// TwinCAT 3 PLC project SSP_M_EGB_v1
// ProgramVersion: 3.1.4024.0
// libraries:
//   EfficientIO Communicator, * (EfficientIO)
//   EfficientIO Energy Basic, * (EfficientIO)
//   Lynus Persistent Data V1, * (Lynus AG)
//   Lynus Standards, * (EfficientIO)
//   Tc2_Standard, * (Beckhoff Automation GmbH)
//   Tc2_System, * (Beckhoff Automation GmbH)
//   Tc2_Utilities, * (Beckhoff Automation GmbH)
//   Tc3_IPCDiag, * (Beckhoff Automation GmbH)
//   Tc3_Module, * (Beckhoff Automation GmbH)
// project tree:
//   ENUM/ E_State.TcDUT (not stored)
//   / FastTask.TcTTO, MiddleTask.TcTTO, SlowTask.TcTTO
//   FBs/ FB_EM_Beckhoff_KL3403_T.TcPOU, prg_ReadDeviceName.TcPOU (not stored)
//   POUs/ prgCalc.TcPOU, prgComEffIO.TcPOU, prgEM.TcPOU, prgPersistent.TcPOU, prgRWEffIO.TcPOU, prgVarEffIO.TcPOU (not stored)

CONFIGURATION SSP_M_EGB_v1
    RESOURCE PLC ON TwinCAT3
        TASK FastTask(INTERVAL := T#10ms, PRIORITY := 21);
        TASK MiddleTask(INTERVAL := T#10ms, PRIORITY := 23);
        TASK SlowTask(INTERVAL := T#10ms, PRIORITY := 22);
        PROGRAM prgRWEffIO WITH FastTask : prgRWEffIO;
        PROGRAM prgVarEffIO WITH FastTask : prgVarEffIO;
        PROGRAM prgPersistent WITH MiddleTask : prgPersistent;
        PROGRAM prgEM WITH MiddleTask : prgEM;
        PROGRAM prgCalc WITH MiddleTask : prgCalc;
        PROGRAM prgComEffIO WITH SlowTask : prgComEffIO;
    END_RESOURCE
END_CONFIGURATION

// ---- POUs/prgRWEffIO.TcPOU
PROGRAM prgRWEffIO
VAR
	fbRW1		: FB_ReadWrite_V2;
	fbRW2		: FB_ReadWrite;
	fbRW3		: FB_ReadWrite;
END_VAR

fbRW1(	eUploadType := eSelectDataUploadType.e_Change_noIntervall,
		bBusy=> , 
		bError=> , 
		udiErrorCodeOut=> , 
		eErrorReadWrite_Out=> );

fbRW2();
		
fbRW3();

END_PROGRAM

// ---- POUs/prgPersistent.TcPOU
PROGRAM prgPersistent
VAR
	fbUSV		: FB_WritePersistentData_CX81xx;
	
	fb_Reboot		: NT_reboot;
	m_Reboot		: BOOL:=FALSE;
END_VAR

fbUSV(
	eSaveModeData:= eUSVSaveMode.eSaveWhenPowerfail, 
	bLoadPersistentDataOk=> , 
	bPowerFailDetect=> , 
	bError=> , 
	bySaveProcess=> , 
	dwStorageLast24h=> , 
	udiErrorCode=> );
	
	
fb_Reboot(	netid := '',
			delay := 2,
			start := m_Reboot);

END_PROGRAM

// ---- POUs/prgEM.TcPOU
PROGRAM prgEM
VAR	
	fbKBusState		: FB_K_Bus_State;
	
	fbEM1			: FB_EM_Beckhoff_KL3403_T;
	fbEM1Counter	: FB_EnergyCounter;
	
	fbEM2			: FB_EM_Beckhoff_KL3403_T;
	fbEM2Counter	: FB_EnergyCounter;
	
	fbEM3			: FB_EM_Beckhoff_KL3403_T;
	fbEM3Counter	: FB_EnergyCounter;
	
	fbEM4			: FB_EM_Beckhoff_KL3403_T;
	fbEM4Counter	: FB_EnergyCounter;
	
	fbEM5			: FB_EM_Beckhoff_KL3403_T;
	fbEM5Counter	: FB_EnergyCounter;
	
	fbEM6			: FB_EM_Beckhoff_KL3403_T;
	fbEM6Counter	: FB_EnergyCounter;
	
	fbEM7			: FB_EM_Beckhoff_KL3403_T;
	fbEM7Counter	: FB_EnergyCounter;
	
	fbEM8			: FB_EM_Beckhoff_KL3403_T;
	fbEM8Counter	: FB_EnergyCounter;
	
	fbEM9			: FB_EM_Beckhoff_KL3403_T;
	fbEM9Counter	: FB_EnergyCounter;

	//EM1 (CEE32 3phase Measurement)
	lr_RealPower_EM1		: LREAL;					//{#lynus.ag#()}
	lr_ApparentPower_EM1	: LREAL;					//{#lynus.ag#()}
	lr_ReactivePower_EM1	: LREAL;					//{#lynus.ag#()}
	lr_Frequency_EM1		: LREAL;					//{#lynus.ag#()}
    lr_RealPower_EM1_L1		: LREAL;					//{#lynus.ag#()}
    lr_RealPower_EM1_L2		: LREAL;					//{#lynus.ag#()}
    lr_RealPower_EM1_L3		: LREAL;					//{#lynus.ag#()}
	lr_Powerfactor_EM1_L1	: LREAL;					//{#lynus.ag#()}
	lr_Powerfactor_EM1_L2	: LREAL;					//{#lynus.ag#()}
	lr_Powerfactor_EM1_L3	: LREAL;					//{#lynus.ag#()}
	lr_ApparentPower_EM1_L1	: LREAL;					//{#lynus.ag#()}
    lr_ApparentPower_EM1_L2	: LREAL;					//{#lynus.ag#()}
    lr_ApparentPower_EM1_L3	: LREAL;					//{#lynus.ag#()}
	lr_ReactivePower_EM1_L1	: LREAL;					//{#lynus.ag#()}
    lr_ReactivePower_EM1_L2	: LREAL;					//{#lynus.ag#()}
    lr_ReactivePower_EM1_L3	: LREAL;					//{#lynus.ag#()}
	lr_Voltage_EM1_L1N		: LREAL;					//{#lynus.ag#()}
	lr_Voltage_EM1_L2N		: LREAL;					//{#lynus.ag#()}
	lr_Voltage_EM1_L3N		: LREAL;					//{#lynus.ag#()}
	lr_Voltage_EM1_L1L2		: LREAL;					//{#lynus.ag#()}
	lr_Voltage_EM1_L2L3		: LREAL;					//{#lynus.ag#()}
	lr_Voltage_EM1_L3L1		: LREAL;					//{#lynus.ag#()}
 	lr_Current_EM1_L1		: LREAL;					//{#lynus.ag#()}
	lr_Current_EM1_L2		: LREAL;					//{#lynus.ag#()}
	lr_Current_EM1_L3		: LREAL;					//{#lynus.ag#()}

    //EM2 (CEE32 3phase Measurement)
	lr_RealPower_EM2		: LREAL;					//{#lynus.ag#()}
	lr_ApparentPower_EM2	: LREAL;					//{#lynus.ag#()}
	lr_ReactivePower_EM2	: LREAL;					//{#lynus.ag#()}
	lr_Frequency_EM2		: LREAL;					//{#lynus.ag#()}
    lr_RealPower_EM2_L1		: LREAL;					//{#lynus.ag#()}
    lr_RealPower_EM2_L2		: LREAL;					//{#lynus.ag#()}
    lr_RealPower_EM2_L3		: LREAL;					//{#lynus.ag#()}
	lr_Powerfactor_EM2_L1	: LREAL;					//{#lynus.ag#()}
	lr_Powerfactor_EM2_L2	: LREAL;					//{#lynus.ag#()}
	lr_Powerfactor_EM2_L3	: LREAL;					//{#lynus.ag#()}
	lr_ApparentPower_EM2_L1	: LREAL;					//{#lynus.ag#()}
    lr_ApparentPower_EM2_L2	: LREAL;					//{#lynus.ag#()}
    lr_ApparentPower_EM2_L3	: LREAL;					//{#lynus.ag#()}
	lr_ReactivePower_EM2_L1	: LREAL;					//{#lynus.ag#()}
    lr_ReactivePower_EM2_L2	: LREAL;					//{#lynus.ag#()}
    lr_ReactivePower_EM2_L3	: LREAL;					//{#lynus.ag#()}
	lr_Voltage_EM2_L1N		: LREAL;					//{#lynus.ag#()}
	lr_Voltage_EM2_L2N		: LREAL;					//{#lynus.ag#()}
	lr_Voltage_EM2_L3N		: LREAL;					//{#lynus.ag#()}
	lr_Voltage_EM2_L1L2		: LREAL;					//{#lynus.ag#()}
	lr_Voltage_EM2_L2L3		: LREAL;					//{#lynus.ag#()}
	lr_Voltage_EM2_L3L1		: LREAL;					//{#lynus.ag#()}
 	lr_Current_EM2_L1		: LREAL;					//{#lynus.ag#()}
	lr_Current_EM2_L2		: LREAL;					//{#lynus.ag#()}
	lr_Current_EM2_L3		: LREAL;					//{#lynus.ag#()}
	
    //EM3 (CEE32 3phase Measurement)
	lr_RealPower_EM3		: LREAL;					//{#lynus.ag#()}
	lr_ApparentPower_EM3	: LREAL;					//{#lynus.ag#()}
	lr_ReactivePower_EM3	: LREAL;					//{#lynus.ag#()}
	lr_Frequency_EM3		: LREAL;					//{#lynus.ag#()}
    lr_RealPower_EM3_L1		: LREAL;					//{#lynus.ag#()}
    lr_RealPower_EM3_L2		: LREAL;					//{#lynus.ag#()}
    lr_RealPower_EM3_L3		: LREAL;					//{#lynus.ag#()}
	lr_Powerfactor_EM3_L1	: LREAL;					//{#lynus.ag#()}
	lr_Powerfactor_EM3_L2	: LREAL;					//{#lynus.ag#()}
	lr_Powerfactor_EM3_L3	: LREAL;					//{#lynus.ag#()}
	lr_ApparentPower_EM3_L1	: LREAL;					//{#lynus.ag#()}
    lr_ApparentPower_EM3_L2	: LREAL;					//{#lynus.ag#()}
    lr_ApparentPower_EM3_L3	: LREAL;					//{#lynus.ag#()}
	lr_ReactivePower_EM3_L1	: LREAL;					//{#lynus.ag#()}
    lr_ReactivePower_EM3_L2	: LREAL;					//{#lynus.ag#()}
    lr_ReactivePower_EM3_L3	: LREAL;					//{#lynus.ag#()}
	lr_Voltage_EM3_L1N		: LREAL;					//{#lynus.ag#()}
	lr_Voltage_EM3_L2N		: LREAL;					//{#lynus.ag#()}
	lr_Voltage_EM3_L3N		: LREAL;					//{#lynus.ag#()}
	lr_Voltage_EM3_L1L2		: LREAL;					//{#lynus.ag#()}
	lr_Voltage_EM3_L2L3		: LREAL;					//{#lynus.ag#()}
	lr_Voltage_EM3_L3L1		: LREAL;					//{#lynus.ag#()}
 	lr_Current_EM3_L1		: LREAL;					//{#lynus.ag#()}
	lr_Current_EM3_L2		: LREAL;					//{#lynus.ag#()}
	lr_Current_EM3_L3		: LREAL;					//{#lynus.ag#()}

    //EM4 (CEE32 3phase Measurement)
	lr_RealPower_EM4		: LREAL;					//{#lynus.ag#()}
	lr_ApparentPower_EM4	: LREAL;					//{#lynus.ag#()}
	lr_ReactivePower_EM4	: LREAL;					//{#lynus.ag#()}
	lr_Frequency_EM4		: LREAL;					//{#lynus.ag#()}
    lr_RealPower_EM4_L1		: LREAL;					//{#lynus.ag#()}
    lr_RealPower_EM4_L2		: LREAL;					//{#lynus.ag#()}
    lr_RealPower_EM4_L3		: LREAL;					//{#lynus.ag#()}
	lr_Powerfactor_EM4_L1	: LREAL;					//{#lynus.ag#()}
	lr_Powerfactor_EM4_L2	: LREAL;					//{#lynus.ag#()}
	lr_Powerfactor_EM4_L3	: LREAL;					//{#lynus.ag#()}
	lr_ApparentPower_EM4_L1	: LREAL;					//{#lynus.ag#()}
    lr_ApparentPower_EM4_L2	: LREAL;					//{#lynus.ag#()}
    lr_ApparentPower_EM4_L3	: LREAL;					//{#lynus.ag#()}
	lr_ReactivePower_EM4_L1	: LREAL;					//{#lynus.ag#()}
    lr_ReactivePower_EM4_L2	: LREAL;					//{#lynus.ag#()}
    lr_ReactivePower_EM4_L3	: LREAL;					//{#lynus.ag#()}
	lr_Voltage_EM4_L1N		: LREAL;					//{#lynus.ag#()}
	lr_Voltage_EM4_L2N		: LREAL;					//{#lynus.ag#()}
	lr_Voltage_EM4_L3N		: LREAL;					//{#lynus.ag#()}
	lr_Voltage_EM4_L1L2		: LREAL;					//{#lynus.ag#()}
	lr_Voltage_EM4_L2L3		: LREAL;					//{#lynus.ag#()}
	lr_Voltage_EM4_L3L1		: LREAL;					//{#lynus.ag#()}
 	lr_Current_EM4_L1		: LREAL;					//{#lynus.ag#()}
	lr_Current_EM4_L2		: LREAL;					//{#lynus.ag#()}
	lr_Current_EM4_L3		: LREAL;					//{#lynus.ag#()}

    //EM5 (CEE32 3phase Measurement)
	lr_RealPower_EM5		: LREAL;					//{#lynus.ag#()}
	lr_ApparentPower_EM5	: LREAL;					//{#lynus.ag#()}
	lr_ReactivePower_EM5	: LREAL;					//{#lynus.ag#()}
	lr_Frequency_EM5		: LREAL;					//{#lynus.ag#()}
    lr_RealPower_EM5_L1		: LREAL;					//{#lynus.ag#()}
    lr_RealPower_EM5_L2		: LREAL;					//{#lynus.ag#()}
    lr_RealPower_EM5_L3		: LREAL;					//{#lynus.ag#()}
	lr_Powerfactor_EM5_L1	: LREAL;					//{#lynus.ag#()}
	lr_Powerfactor_EM5_L2	: LREAL;					//{#lynus.ag#()}
	lr_Powerfactor_EM5_L3	: LREAL;					//{#lynus.ag#()}
	lr_ApparentPower_EM5_L1	: LREAL;					//{#lynus.ag#()}
    lr_ApparentPower_EM5_L2	: LREAL;					//{#lynus.ag#()}
    lr_ApparentPower_EM5_L3	: LREAL;					//{#lynus.ag#()}
	lr_ReactivePower_EM5_L1	: LREAL;					//{#lynus.ag#()}
    lr_ReactivePower_EM5_L2	: LREAL;					//{#lynus.ag#()}
    lr_ReactivePower_EM5_L3	: LREAL;					//{#lynus.ag#()}
	lr_Voltage_EM5_L1N		: LREAL;					//{#lynus.ag#()}
	lr_Voltage_EM5_L2N		: LREAL;					//{#lynus.ag#()}
	lr_Voltage_EM5_L3N		: LREAL;					//{#lynus.ag#()}
	lr_Voltage_EM5_L1L2		: LREAL;					//{#lynus.ag#()}
	lr_Voltage_EM5_L2L3		: LREAL;					//{#lynus.ag#()}
	lr_Voltage_EM5_L3L1		: LREAL;					//{#lynus.ag#()}
 	lr_Current_EM5_L1		: LREAL;					//{#lynus.ag#()}
	lr_Current_EM5_L2		: LREAL;					//{#lynus.ag#()}
	lr_Current_EM5_L3		: LREAL;					//{#lynus.ag#()}

    //EM6 (CEE32 3phase Measurement)
	lr_RealPower_EM6		: LREAL;					//{#lynus.ag#()}
	lr_ApparentPower_EM6	: LREAL;					//{#lynus.ag#()}
	lr_ReactivePower_EM6	: LREAL;					//{#lynus.ag#()}
	lr_Frequency_EM6		: LREAL;					//{#lynus.ag#()}
    lr_RealPower_EM6_L1		: LREAL;					//{#lynus.ag#()}
    lr_RealPower_EM6_L2		: LREAL;					//{#lynus.ag#()}
    lr_RealPower_EM6_L3		: LREAL;					//{#lynus.ag#()}
	lr_Powerfactor_EM6_L1	: LREAL;					//{#lynus.ag#()}
	lr_Powerfactor_EM6_L2	: LREAL;					//{#lynus.ag#()}
	lr_Powerfactor_EM6_L3	: LREAL;					//{#lynus.ag#()}
	lr_ApparentPower_EM6_L1	: LREAL;					//{#lynus.ag#()}
    lr_ApparentPower_EM6_L2	: LREAL;					//{#lynus.ag#()}
    lr_ApparentPower_EM6_L3	: LREAL;					//{#lynus.ag#()}
	lr_ReactivePower_EM6_L1	: LREAL;					//{#lynus.ag#()}
    lr_ReactivePower_EM6_L2	: LREAL;					//{#lynus.ag#()}
    lr_ReactivePower_EM6_L3	: LREAL;					//{#lynus.ag#()}
	lr_Voltage_EM6_L1N		: LREAL;					//{#lynus.ag#()}
	lr_Voltage_EM6_L2N		: LREAL;					//{#lynus.ag#()}
	lr_Voltage_EM6_L3N		: LREAL;					//{#lynus.ag#()}
	lr_Voltage_EM6_L1L2		: LREAL;					//{#lynus.ag#()}
	lr_Voltage_EM6_L2L3		: LREAL;					//{#lynus.ag#()}
	lr_Voltage_EM6_L3L1		: LREAL;					//{#lynus.ag#()}
 	lr_Current_EM6_L1		: LREAL;					//{#lynus.ag#()}
	lr_Current_EM6_L2		: LREAL;					//{#lynus.ag#()}
	lr_Current_EM6_L3		: LREAL;					//{#lynus.ag#()}

    //EM7 (CEE32 3phase Measurement)
	lr_RealPower_EM7		: LREAL;					//{#lynus.ag#()}
	lr_ApparentPower_EM7	: LREAL;					//{#lynus.ag#()}
	lr_ReactivePower_EM7	: LREAL;					//{#lynus.ag#()}
	lr_Frequency_EM7		: LREAL;					//{#lynus.ag#()}
    lr_RealPower_EM7_L1		: LREAL;					//{#lynus.ag#()}
    lr_RealPower_EM7_L2		: LREAL;					//{#lynus.ag#()}
    lr_RealPower_EM7_L3		: LREAL;					//{#lynus.ag#()}
	lr_Powerfactor_EM7_L1	: LREAL;					//{#lynus.ag#()}
	lr_Powerfactor_EM7_L2	: LREAL;					//{#lynus.ag#()}
	lr_Powerfactor_EM7_L3	: LREAL;					//{#lynus.ag#()}
	lr_ApparentPower_EM7_L1	: LREAL;					//{#lynus.ag#()}
    lr_ApparentPower_EM7_L2	: LREAL;					//{#lynus.ag#()}
    lr_ApparentPower_EM7_L3	: LREAL;					//{#lynus.ag#()}
	lr_ReactivePower_EM7_L1	: LREAL;					//{#lynus.ag#()}
    lr_ReactivePower_EM7_L2	: LREAL;					//{#lynus.ag#()}
    lr_ReactivePower_EM7_L3	: LREAL;					//{#lynus.ag#()}
	lr_Voltage_EM7_L1N		: LREAL;					//{#lynus.ag#()}
	lr_Voltage_EM7_L2N		: LREAL;					//{#lynus.ag#()}
	lr_Voltage_EM7_L3N		: LREAL;					//{#lynus.ag#()}
	lr_Voltage_EM7_L1L2		: LREAL;					//{#lynus.ag#()}
	lr_Voltage_EM7_L2L3		: LREAL;					//{#lynus.ag#()}
	lr_Voltage_EM7_L3L1		: LREAL;					//{#lynus.ag#()}
 	lr_Current_EM7_L1		: LREAL;					//{#lynus.ag#()}
	lr_Current_EM7_L2		: LREAL;					//{#lynus.ag#()}
	lr_Current_EM7_L3		: LREAL;					//{#lynus.ag#()}

    //EM8 (CEE32 3phase Measurement)
	lr_RealPower_EM8		: LREAL;					//{#lynus.ag#()}
	lr_ApparentPower_EM8	: LREAL;					//{#lynus.ag#()}
	lr_ReactivePower_EM8	: LREAL;					//{#lynus.ag#()}
	lr_Frequency_EM8		: LREAL;					//{#lynus.ag#()}
    lr_RealPower_EM8_L1		: LREAL;					//{#lynus.ag#()}
    lr_RealPower_EM8_L2		: LREAL;					//{#lynus.ag#()}
    lr_RealPower_EM8_L3		: LREAL;					//{#lynus.ag#()}
	lr_Powerfactor_EM8_L1	: LREAL;					//{#lynus.ag#()}
	lr_Powerfactor_EM8_L2	: LREAL;					//{#lynus.ag#()}
	lr_Powerfactor_EM8_L3	: LREAL;					//{#lynus.ag#()}
	lr_ApparentPower_EM8_L1	: LREAL;					//{#lynus.ag#()}
    lr_ApparentPower_EM8_L2	: LREAL;					//{#lynus.ag#()}
    lr_ApparentPower_EM8_L3	: LREAL;					//{#lynus.ag#()}
	lr_ReactivePower_EM8_L1	: LREAL;					//{#lynus.ag#()}
    lr_ReactivePower_EM8_L2	: LREAL;					//{#lynus.ag#()}
    lr_ReactivePower_EM8_L3	: LREAL;					//{#lynus.ag#()}
	lr_Voltage_EM8_L1N		: LREAL;					//{#lynus.ag#()}
	lr_Voltage_EM8_L2N		: LREAL;					//{#lynus.ag#()}
	lr_Voltage_EM8_L3N		: LREAL;					//{#lynus.ag#()}
	lr_Voltage_EM8_L1L2		: LREAL;					//{#lynus.ag#()}
	lr_Voltage_EM8_L2L3		: LREAL;					//{#lynus.ag#()}
	lr_Voltage_EM8_L3L1		: LREAL;					//{#lynus.ag#()}
 	lr_Current_EM8_L1		: LREAL;					//{#lynus.ag#()}
	lr_Current_EM8_L2		: LREAL;					//{#lynus.ag#()}
	lr_Current_EM8_L3		: LREAL;					//{#lynus.ag#()}

    //EM9 (CEE32 3phase Measurement)
	lr_RealPower_EM9		: LREAL;					//{#lynus.ag#()}
	lr_ApparentPower_EM9	: LREAL;					//{#lynus.ag#()}
	lr_ReactivePower_EM9	: LREAL;					//{#lynus.ag#()}
	lr_Frequency_EM9		: LREAL;					//{#lynus.ag#()}
    lr_RealPower_EM9_L1		: LREAL;					//{#lynus.ag#()}
    lr_RealPower_EM9_L2		: LREAL;					//{#lynus.ag#()}
    lr_RealPower_EM9_L3		: LREAL;					//{#lynus.ag#()}
	lr_Powerfactor_EM9_L1	: LREAL;					//{#lynus.ag#()}
	lr_Powerfactor_EM9_L2	: LREAL;					//{#lynus.ag#()}
	lr_Powerfactor_EM9_L3	: LREAL;					//{#lynus.ag#()}
	lr_ApparentPower_EM9_L1	: LREAL;					//{#lynus.ag#()}
    lr_ApparentPower_EM9_L2	: LREAL;					//{#lynus.ag#()}
    lr_ApparentPower_EM9_L3	: LREAL;					//{#lynus.ag#()}
	lr_ReactivePower_EM9_L1	: LREAL;					//{#lynus.ag#()}
    lr_ReactivePower_EM9_L2	: LREAL;					//{#lynus.ag#()}
    lr_ReactivePower_EM9_L3	: LREAL;					//{#lynus.ag#()}
	lr_Voltage_EM9_L1N		: LREAL;					//{#lynus.ag#()}
	lr_Voltage_EM9_L2N		: LREAL;					//{#lynus.ag#()}
	lr_Voltage_EM9_L3N		: LREAL;					//{#lynus.ag#()}
	lr_Voltage_EM9_L1L2		: LREAL;					//{#lynus.ag#()}
	lr_Voltage_EM9_L2L3		: LREAL;					//{#lynus.ag#()}
	lr_Voltage_EM9_L3L1		: LREAL;					//{#lynus.ag#()}
 	lr_Current_EM9_L1		: LREAL;					//{#lynus.ag#()}
	lr_Current_EM9_L2		: LREAL;					//{#lynus.ag#()}
	lr_Current_EM9_L3		: LREAL;					//{#lynus.ag#()}
END_VAR

VAR PERSISTENT
	lr_EnergyCounter_EM1	: LREAL;					//{#lynus.ag#()}
	lr_EnergyCounter_EM2	: LREAL;					//{#lynus.ag#()}
    lr_EnergyCounter_EM3	: LREAL;					//{#lynus.ag#()}
    lr_EnergyCounter_EM4	: LREAL;					//{#lynus.ag#()}
    lr_EnergyCounter_EM5	: LREAL;					//{#lynus.ag#()}
    lr_EnergyCounter_EM6	: LREAL;					//{#lynus.ag#()}
    lr_EnergyCounter_EM7	: LREAL;					//{#lynus.ag#()}
    lr_EnergyCounter_EM8	: LREAL;					//{#lynus.ag#()}
    lr_EnergyCounter_EM9	: LREAL;					//{#lynus.ag#()}
END_VAR

fbKBusState(	uiKBusState_OUT=> , 
				b_Kbus_notOk=> , 
				word_ErrorCount=> );

//EM1 (CEE32 3phase Measurement)
fbEM1(
	bEnable:= TRUE, 
	bChannel1Invers:= FALSE,
	bChannel2Invers:= FALSE,
	bChannel3Invers:= FALSE,
	uiCurrentTransformerRatioL1:= 35, 
	uiCurrentTransformerRatioL2:= 35, 
	uiCurrentTransformerRatioL3:= 35, 
	uiKBusState_IN:= fbKBusState.uiKBusState_OUT, 
	stDataEMPower=> , 
	stDataEMCounter=> , 
	stDataEMPowerRealTime=> , 
	stDataEMCounterRealTime=> , 
	diNrOfEM_OUT=> );

lr_RealPower_EM1 := fbEM1.stDataEMPower.lrPowerTotal;
lr_ApparentPower_EM1 := fbEM1.stDataEMPower.lrApparentPowerTotal;
lr_ReactivePower_EM1 := fbEM1.stDataEMPower.lrReactivePowerTotal;
lr_Frequency_EM1 := fbEM1.stDataEMPower.lrFrequency;
lr_RealPower_EM1_L1 := fbEM1.stDataEMPower.lrPowerL1;
lr_RealPower_EM1_L2 := fbEM1.stDataEMPower.lrPowerL2;
lr_RealPower_EM1_L3 := fbEM1.stDataEMPower.lrPowerL3;
lr_Voltage_EM1_L1N := fbEM1.stDataEMPower.lrVoltageL1N;
lr_Voltage_EM1_L2N := fbEM1.stDataEMPower.lrVoltageL2N;
lr_Voltage_EM1_L3N := fbEM1.stDataEMPower.lrVoltageL3N;
lr_Voltage_EM1_L1L2 := fbEM1.stDataEMPower.lrVoltageL1L2;
lr_Voltage_EM1_L2L3 := fbEM1.stDataEMPower.lrVoltageL2L3;
lr_Voltage_EM1_L3L1 := fbEM1.stDataEMPower.lrVoltageL3L1;
lr_Current_EM1_L1 := fbEM1.stDataEMPower.lrCurrentL1;
lr_Current_EM1_L2 := fbEM1.stDataEMPower.lrCurrentL2;
lr_Current_EM1_L3 := fbEM1.stDataEMPower.lrCurrentL3;
lr_Powerfactor_EM1_L1 := fbEM1.lrPowerfactorL1;
lr_Powerfactor_EM1_L2 := fbEM1.lrPowerfactorL2;
lr_Powerfactor_EM1_L3 := fbEM1.lrPowerfactorL3;
(*
lr_ApparentPower_EM1_L1 := fbEM1.lrApparentPowerL1;
lr_ApparentPower_EM1_L2 := fbEM1.lrApparentPowerL2;
lr_ApparentPower_EM1_L3 := fbEM1.lrApparentPowerL3;
lr_ReactivePower_EM1_L1 := fbEM1.lrReactivePowerL1;
lr_ReactivePower_EM1_L2 := fbEM1.lrReactivePowerL2;
lr_ReactivePower_EM1_L3 := fbEM1.lrReactivePowerL3;
*)
fbEM1Counter(
	byActiveTariff:= 1, 
	lrPowerInput:= lr_RealPower_EM1, 
	lrTotalCounterEnergy_Consumption=> , 
	lrTotalCounterEnergy_Production=> , 
	lrCounterEnergyT1_Consumption=> , 
	lrCounterEnergyT2_Consumption=> , 
	lrCounterEnergyT1_Production=> , 
	lrCounterEnergyT2_Production=> );
	
IF fbEM1Counter.lrTotalCounterEnergy_Consumption > lr_EnergyCounter_EM1 THEN  	
	lr_EnergyCounter_EM1 := fbEM1Counter.lrTotalCounterEnergy_Consumption;
END_IF


//EM2 (CEE32 3phase Measurement)
fbEM2(
	bEnable:= TRUE, 
	bChannel1Invers:= FALSE,
	bChannel2Invers:= FALSE,
	bChannel3Invers:= FALSE,
	uiCurrentTransformerRatioL1:= 35, 
	uiCurrentTransformerRatioL2:= 35, 
	uiCurrentTransformerRatioL3:= 35, 
	uiKBusState_IN:= fbKBusState.uiKBusState_OUT, 
	stDataEMPower=> , 
	stDataEMCounter=> , 
	stDataEMPowerRealTime=> , 
	stDataEMCounterRealTime=> , 
	diNrOfEM_OUT=> );

lr_RealPower_EM2 := fbEM2.stDataEMPower.lrPowerTotal;
lr_ApparentPower_EM2 := fbEM2.stDataEMPower.lrApparentPowerTotal;
lr_ReactivePower_EM2 := fbEM2.stDataEMPower.lrReactivePowerTotal;
lr_Frequency_EM2 := fbEM2.stDataEMPower.lrFrequency;
lr_RealPower_EM2_L1 := fbEM2.stDataEMPower.lrPowerL1;
lr_RealPower_EM2_L2 := fbEM2.stDataEMPower.lrPowerL2;
lr_RealPower_EM2_L3 := fbEM2.stDataEMPower.lrPowerL3;
lr_Voltage_EM2_L1N := fbEM2.stDataEMPower.lrVoltageL1N;
lr_Voltage_EM2_L2N := fbEM2.stDataEMPower.lrVoltageL2N;
lr_Voltage_EM2_L3N := fbEM2.stDataEMPower.lrVoltageL3N;
lr_Voltage_EM2_L1L2 := fbEM2.stDataEMPower.lrVoltageL1L2;
lr_Voltage_EM2_L2L3 := fbEM2.stDataEMPower.lrVoltageL2L3;
lr_Voltage_EM2_L3L1 := fbEM2.stDataEMPower.lrVoltageL3L1;
lr_Current_EM2_L1 := fbEM2.stDataEMPower.lrCurrentL1;
lr_Current_EM2_L2 := fbEM2.stDataEMPower.lrCurrentL2;
lr_Current_EM2_L3 := fbEM2.stDataEMPower.lrCurrentL3;
lr_Powerfactor_EM2_L1 := fbEM2.lrPowerfactorL1;
lr_Powerfactor_EM2_L2 := fbEM2.lrPowerfactorL2;
lr_Powerfactor_EM2_L3 := fbEM2.lrPowerfactorL3;
(*
lr_ApparentPower_EM2_L1 := fbEM2.lrApparentPowerL1;
lr_ApparentPower_EM2_L2 := fbEM2.lrApparentPowerL2;
lr_ApparentPower_EM2_L3 := fbEM2.lrApparentPowerL3;
lr_ReactivePower_EM2_L1 := fbEM2.lrReactivePowerL1;
lr_ReactivePower_EM2_L2 := fbEM2.lrReactivePowerL2;
lr_ReactivePower_EM2_L3 := fbEM2.lrReactivePowerL3;
*)
fbEM2Counter(
	byActiveTariff:= 1, 
	lrPowerInput:= lr_RealPower_EM2, 
	lrTotalCounterEnergy_Consumption=> , 
	lrTotalCounterEnergy_Production=> , 
	lrCounterEnergyT1_Consumption=> , 
	lrCounterEnergyT2_Consumption=> , 
	lrCounterEnergyT1_Production=> , 
	lrCounterEnergyT2_Production=> );
	
IF fbEM2Counter.lrTotalCounterEnergy_Consumption > lr_EnergyCounter_EM2 THEN  	
	lr_EnergyCounter_EM2 := fbEM2Counter.lrTotalCounterEnergy_Consumption;
END_IF

//EM3 (CEE32 3phase Measurement)
fbEM3(
	bEnable:= TRUE, 
	bChannel1Invers:= FALSE,
	bChannel2Invers:= FALSE,
	bChannel3Invers:= FALSE,
	uiCurrentTransformerRatioL1:= 35, 
	uiCurrentTransformerRatioL2:= 35, 
	uiCurrentTransformerRatioL3:= 35, 
	uiKBusState_IN:= fbKBusState.uiKBusState_OUT, 
	stDataEMPower=> , 
	stDataEMCounter=> , 
	stDataEMPowerRealTime=> , 
	stDataEMCounterRealTime=> , 
	diNrOfEM_OUT=> );

lr_RealPower_EM3 := fbEM3.stDataEMPower.lrPowerTotal;
lr_ApparentPower_EM3 := fbEM3.stDataEMPower.lrApparentPowerTotal;
lr_ReactivePower_EM3 := fbEM3.stDataEMPower.lrReactivePowerTotal;
lr_Frequency_EM3 := fbEM3.stDataEMPower.lrFrequency;
lr_RealPower_EM3_L1 := fbEM3.stDataEMPower.lrPowerL1;
lr_RealPower_EM3_L2 := fbEM3.stDataEMPower.lrPowerL2;
lr_RealPower_EM3_L3 := fbEM3.stDataEMPower.lrPowerL3;
lr_Voltage_EM3_L1N := fbEM3.stDataEMPower.lrVoltageL1N;
lr_Voltage_EM3_L2N := fbEM3.stDataEMPower.lrVoltageL2N;
lr_Voltage_EM3_L3N := fbEM3.stDataEMPower.lrVoltageL3N;
lr_Voltage_EM3_L1L2 := fbEM3.stDataEMPower.lrVoltageL1L2;
lr_Voltage_EM3_L2L3 := fbEM3.stDataEMPower.lrVoltageL2L3;
lr_Voltage_EM3_L3L1 := fbEM3.stDataEMPower.lrVoltageL3L1;
lr_Current_EM3_L1 := fbEM3.stDataEMPower.lrCurrentL1;
lr_Current_EM3_L2 := fbEM3.stDataEMPower.lrCurrentL2;
lr_Current_EM3_L3 := fbEM3.stDataEMPower.lrCurrentL3;
lr_Powerfactor_EM3_L1 := fbEM3.lrPowerfactorL1;
lr_Powerfactor_EM3_L2 := fbEM3.lrPowerfactorL2;
lr_Powerfactor_EM3_L3 := fbEM3.lrPowerfactorL3;
(*
lr_ApparentPower_EM3_L1 := fbEM3.lrApparentPowerL1;
lr_ApparentPower_EM3_L2 := fbEM3.lrApparentPowerL2;
lr_ApparentPower_EM3_L3 := fbEM3.lrApparentPowerL3;
lr_ReactivePower_EM3_L1 := fbEM3.lrReactivePowerL1;
lr_ReactivePower_EM3_L2 := fbEM3.lrReactivePowerL2;
lr_ReactivePower_EM3_L3 := fbEM3.lrReactivePowerL3;
*)
fbEM3Counter(
	byActiveTariff:= 1, 
	lrPowerInput:= lr_RealPower_EM3, 
	lrTotalCounterEnergy_Consumption=> , 
	lrTotalCounterEnergy_Production=> , 
	lrCounterEnergyT1_Consumption=> , 
	lrCounterEnergyT2_Consumption=> , 
	lrCounterEnergyT1_Production=> , 
	lrCounterEnergyT2_Production=> );
	
IF fbEM3Counter.lrTotalCounterEnergy_Consumption > lr_EnergyCounter_EM3 THEN  	
	lr_EnergyCounter_EM3 := fbEM3Counter.lrTotalCounterEnergy_Consumption;
END_IF

//EM4 (CEE32 3phase Measurement)
fbEM4(
	bEnable:= TRUE, 
	bChannel1Invers:= FALSE,
	bChannel2Invers:= FALSE,
	bChannel3Invers:= FALSE,
	uiCurrentTransformerRatioL1:= 35, 
	uiCurrentTransformerRatioL2:= 35, 
	uiCurrentTransformerRatioL3:= 35, 
	uiKBusState_IN:= fbKBusState.uiKBusState_OUT, 
	stDataEMPower=> , 
	stDataEMCounter=> , 
	stDataEMPowerRealTime=> , 
	stDataEMCounterRealTime=> , 
	diNrOfEM_OUT=> );

lr_RealPower_EM4 := fbEM4.stDataEMPower.lrPowerTotal;
lr_ApparentPower_EM4 := fbEM4.stDataEMPower.lrApparentPowerTotal;
lr_ReactivePower_EM4 := fbEM4.stDataEMPower.lrReactivePowerTotal;
lr_Frequency_EM4 := fbEM4.stDataEMPower.lrFrequency;
lr_RealPower_EM4_L1 := fbEM4.stDataEMPower.lrPowerL1;
lr_RealPower_EM4_L2 := fbEM4.stDataEMPower.lrPowerL2;
lr_RealPower_EM4_L3 := fbEM4.stDataEMPower.lrPowerL3;
lr_Voltage_EM4_L1N := fbEM4.stDataEMPower.lrVoltageL1N;
lr_Voltage_EM4_L2N := fbEM4.stDataEMPower.lrVoltageL2N;
lr_Voltage_EM4_L3N := fbEM4.stDataEMPower.lrVoltageL3N;
lr_Voltage_EM4_L1L2 := fbEM4.stDataEMPower.lrVoltageL1L2;
lr_Voltage_EM4_L2L3 := fbEM4.stDataEMPower.lrVoltageL2L3;
lr_Voltage_EM4_L3L1 := fbEM4.stDataEMPower.lrVoltageL3L1;
lr_Current_EM4_L1 := fbEM4.stDataEMPower.lrCurrentL1;
lr_Current_EM4_L2 := fbEM4.stDataEMPower.lrCurrentL2;
lr_Current_EM4_L3 := fbEM4.stDataEMPower.lrCurrentL3;
lr_Powerfactor_EM4_L1 := fbEM4.lrPowerfactorL1;
lr_Powerfactor_EM4_L2 := fbEM4.lrPowerfactorL2;
lr_Powerfactor_EM4_L3 := fbEM4.lrPowerfactorL3;
(*
lr_ApparentPower_EM4_L1 := fbEM4.lrApparentPowerL1;
lr_ApparentPower_EM4_L2 := fbEM4.lrApparentPowerL2;
lr_ApparentPower_EM4_L3 := fbEM4.lrApparentPowerL3;
lr_ReactivePower_EM4_L1 := fbEM4.lrReactivePowerL1;
lr_ReactivePower_EM4_L2 := fbEM4.lrReactivePowerL2;
lr_ReactivePower_EM4_L3 := fbEM4.lrReactivePowerL3;
*)
fbEM4Counter(
	byActiveTariff:= 1, 
	lrPowerInput:= lr_RealPower_EM4, 
	lrTotalCounterEnergy_Consumption=> , 
	lrTotalCounterEnergy_Production=> , 
	lrCounterEnergyT1_Consumption=> , 
	lrCounterEnergyT2_Consumption=> , 
	lrCounterEnergyT1_Production=> , 
	lrCounterEnergyT2_Production=> );
	
IF fbEM4Counter.lrTotalCounterEnergy_Consumption > lr_EnergyCounter_EM4 THEN  	
	lr_EnergyCounter_EM4 := fbEM4Counter.lrTotalCounterEnergy_Consumption;
END_IF

//EM5 (CEE32 3phase Measurement)
fbEM5(
	bEnable:= TRUE, 
	bChannel1Invers:= FALSE,
	bChannel2Invers:= FALSE,
	bChannel3Invers:= FALSE,
	uiCurrentTransformerRatioL1:= 35, 
	uiCurrentTransformerRatioL2:= 35, 
	uiCurrentTransformerRatioL3:= 35, 
	uiKBusState_IN:= fbKBusState.uiKBusState_OUT, 
	stDataEMPower=> , 
	stDataEMCounter=> , 
	stDataEMPowerRealTime=> , 
	stDataEMCounterRealTime=> , 
	diNrOfEM_OUT=> );

lr_RealPower_EM5 := fbEM5.stDataEMPower.lrPowerTotal;
lr_ApparentPower_EM5 := fbEM5.stDataEMPower.lrApparentPowerTotal;
lr_ReactivePower_EM5 := fbEM5.stDataEMPower.lrReactivePowerTotal;
lr_Frequency_EM5 := fbEM5.stDataEMPower.lrFrequency;
lr_RealPower_EM5_L1 := fbEM5.stDataEMPower.lrPowerL1;
lr_RealPower_EM5_L2 := fbEM5.stDataEMPower.lrPowerL2;
lr_RealPower_EM5_L3 := fbEM5.stDataEMPower.lrPowerL3;
lr_Voltage_EM5_L1N := fbEM5.stDataEMPower.lrVoltageL1N;
lr_Voltage_EM5_L2N := fbEM5.stDataEMPower.lrVoltageL2N;
lr_Voltage_EM5_L3N := fbEM5.stDataEMPower.lrVoltageL3N;
lr_Voltage_EM5_L1L2 := fbEM5.stDataEMPower.lrVoltageL1L2;
lr_Voltage_EM5_L2L3 := fbEM5.stDataEMPower.lrVoltageL2L3;
lr_Voltage_EM5_L3L1 := fbEM5.stDataEMPower.lrVoltageL3L1;
lr_Current_EM5_L1 := fbEM5.stDataEMPower.lrCurrentL1;
lr_Current_EM5_L2 := fbEM5.stDataEMPower.lrCurrentL2;
lr_Current_EM5_L3 := fbEM5.stDataEMPower.lrCurrentL3;
lr_Powerfactor_EM5_L1 := fbEM5.lrPowerfactorL1;
lr_Powerfactor_EM5_L2 := fbEM5.lrPowerfactorL2;
lr_Powerfactor_EM5_L3 := fbEM5.lrPowerfactorL3;
(*
lr_ApparentPower_EM5_L1 := fbEM5.lrApparentPowerL1;
lr_ApparentPower_EM5_L2 := fbEM5.lrApparentPowerL2;
lr_ApparentPower_EM5_L3 := fbEM5.lrApparentPowerL3;
lr_ReactivePower_EM5_L1 := fbEM5.lrReactivePowerL1;
lr_ReactivePower_EM5_L2 := fbEM5.lrReactivePowerL2;
lr_ReactivePower_EM5_L3 := fbEM5.lrReactivePowerL3;
*)
fbEM5Counter(
	byActiveTariff:= 1, 
	lrPowerInput:= lr_RealPower_EM5, 
	lrTotalCounterEnergy_Consumption=> , 
	lrTotalCounterEnergy_Production=> , 
	lrCounterEnergyT1_Consumption=> , 
	lrCounterEnergyT2_Consumption=> , 
	lrCounterEnergyT1_Production=> , 
	lrCounterEnergyT2_Production=> );
	
IF fbEM5Counter.lrTotalCounterEnergy_Consumption > lr_EnergyCounter_EM5 THEN  	
	lr_EnergyCounter_EM5 := fbEM5Counter.lrTotalCounterEnergy_Consumption;
END_IF

//EM6 (CEE32 3phase Measurement)
fbEM6(
	bEnable:= TRUE, 
	bChannel1Invers:= FALSE,
	bChannel2Invers:= FALSE,
	bChannel3Invers:= FALSE,
	uiCurrentTransformerRatioL1:= 35, 
	uiCurrentTransformerRatioL2:= 35, 
	uiCurrentTransformerRatioL3:= 35, 
	uiKBusState_IN:= fbKBusState.uiKBusState_OUT, 
	stDataEMPower=> , 
	stDataEMCounter=> , 
	stDataEMPowerRealTime=> , 
	stDataEMCounterRealTime=> , 
	diNrOfEM_OUT=> );

lr_RealPower_EM6 := fbEM6.stDataEMPower.lrPowerTotal;
lr_ApparentPower_EM6 := fbEM6.stDataEMPower.lrApparentPowerTotal;
lr_ReactivePower_EM6 := fbEM6.stDataEMPower.lrReactivePowerTotal;
lr_Frequency_EM6 := fbEM6.stDataEMPower.lrFrequency;
lr_RealPower_EM6_L1 := fbEM6.stDataEMPower.lrPowerL1;
lr_RealPower_EM6_L2 := fbEM6.stDataEMPower.lrPowerL2;
lr_RealPower_EM6_L3 := fbEM6.stDataEMPower.lrPowerL3;
lr_Voltage_EM6_L1N := fbEM6.stDataEMPower.lrVoltageL1N;
lr_Voltage_EM6_L2N := fbEM6.stDataEMPower.lrVoltageL2N;
lr_Voltage_EM6_L3N := fbEM6.stDataEMPower.lrVoltageL3N;
lr_Voltage_EM6_L1L2 := fbEM6.stDataEMPower.lrVoltageL1L2;
lr_Voltage_EM6_L2L3 := fbEM6.stDataEMPower.lrVoltageL2L3;
lr_Voltage_EM6_L3L1 := fbEM6.stDataEMPower.lrVoltageL3L1;
lr_Current_EM6_L1 := fbEM6.stDataEMPower.lrCurrentL1;
lr_Current_EM6_L2 := fbEM6.stDataEMPower.lrCurrentL2;
lr_Current_EM6_L3 := fbEM6.stDataEMPower.lrCurrentL3;
lr_Powerfactor_EM6_L1 := fbEM6.lrPowerfactorL1;
lr_Powerfactor_EM6_L2 := fbEM6.lrPowerfactorL2;
lr_Powerfactor_EM6_L3 := fbEM6.lrPowerfactorL3;
(*
lr_ApparentPower_EM6_L1 := fbEM6.lrApparentPowerL1;
lr_ApparentPower_EM6_L2 := fbEM6.lrApparentPowerL2;
lr_ApparentPower_EM6_L3 := fbEM6.lrApparentPowerL3;
lr_ReactivePower_EM6_L1 := fbEM6.lrReactivePowerL1;
lr_ReactivePower_EM6_L2 := fbEM6.lrReactivePowerL2;
lr_ReactivePower_EM6_L3 := fbEM6.lrReactivePowerL3;
*)
fbEM6Counter(
	byActiveTariff:= 1, 
	lrPowerInput:= lr_RealPower_EM6, 
	lrTotalCounterEnergy_Consumption=> , 
	lrTotalCounterEnergy_Production=> , 
	lrCounterEnergyT1_Consumption=> , 
	lrCounterEnergyT2_Consumption=> , 
	lrCounterEnergyT1_Production=> , 
	lrCounterEnergyT2_Production=> );
	
IF fbEM6Counter.lrTotalCounterEnergy_Consumption > lr_EnergyCounter_EM6 THEN  	
	lr_EnergyCounter_EM6 := fbEM6Counter.lrTotalCounterEnergy_Consumption;
END_IF

//EM7 (CEE32 3phase Measurement)
fbEM7(
	bEnable:= TRUE, 
	bChannel1Invers:= FALSE,
	bChannel2Invers:= FALSE,
	bChannel3Invers:= FALSE,
	uiCurrentTransformerRatioL1:= 35, 
	uiCurrentTransformerRatioL2:= 35, 
	uiCurrentTransformerRatioL3:= 35, 
	uiKBusState_IN:= fbKBusState.uiKBusState_OUT, 
	stDataEMPower=> , 
	stDataEMCounter=> , 
	stDataEMPowerRealTime=> , 
	stDataEMCounterRealTime=> , 
	diNrOfEM_OUT=> );

lr_RealPower_EM7 := fbEM7.stDataEMPower.lrPowerTotal;
lr_ApparentPower_EM7 := fbEM7.stDataEMPower.lrApparentPowerTotal;
lr_ReactivePower_EM7 := fbEM7.stDataEMPower.lrReactivePowerTotal;
lr_Frequency_EM7 := fbEM7.stDataEMPower.lrFrequency;
lr_RealPower_EM7_L1 := fbEM7.stDataEMPower.lrPowerL1;
lr_RealPower_EM7_L2 := fbEM7.stDataEMPower.lrPowerL2;
lr_RealPower_EM7_L3 := fbEM7.stDataEMPower.lrPowerL3;
lr_Voltage_EM7_L1N := fbEM7.stDataEMPower.lrVoltageL1N;
lr_Voltage_EM7_L2N := fbEM7.stDataEMPower.lrVoltageL2N;
lr_Voltage_EM7_L3N := fbEM7.stDataEMPower.lrVoltageL3N;
lr_Voltage_EM7_L1L2 := fbEM7.stDataEMPower.lrVoltageL1L2;
lr_Voltage_EM7_L2L3 := fbEM7.stDataEMPower.lrVoltageL2L3;
lr_Voltage_EM7_L3L1 := fbEM7.stDataEMPower.lrVoltageL3L1;
lr_Current_EM7_L1 := fbEM7.stDataEMPower.lrCurrentL1;
lr_Current_EM7_L2 := fbEM7.stDataEMPower.lrCurrentL2;
lr_Current_EM7_L3 := fbEM7.stDataEMPower.lrCurrentL3;
lr_Powerfactor_EM7_L1 := fbEM7.lrPowerfactorL1;
lr_Powerfactor_EM7_L2 := fbEM7.lrPowerfactorL2;
lr_Powerfactor_EM7_L3 := fbEM7.lrPowerfactorL3;
(*
lr_ApparentPower_EM7_L1 := fbEM7.lrApparentPowerL1;
lr_ApparentPower_EM7_L2 := fbEM7.lrApparentPowerL2;
lr_ApparentPower_EM7_L3 := fbEM7.lrApparentPowerL3;
lr_ReactivePower_EM7_L1 := fbEM7.lrReactivePowerL1;
lr_ReactivePower_EM7_L2 := fbEM7.lrReactivePowerL2;
lr_ReactivePower_EM7_L3 := fbEM7.lrReactivePowerL3;
*)
fbEM7Counter(
	byActiveTariff:= 1, 
	lrPowerInput:= lr_RealPower_EM7, 
	lrTotalCounterEnergy_Consumption=> , 
	lrTotalCounterEnergy_Production=> , 
	lrCounterEnergyT1_Consumption=> , 
	lrCounterEnergyT2_Consumption=> , 
	lrCounterEnergyT1_Production=> , 
	lrCounterEnergyT2_Production=> );
	
IF fbEM7Counter.lrTotalCounterEnergy_Consumption > lr_EnergyCounter_EM7 THEN  	
	lr_EnergyCounter_EM7 := fbEM7Counter.lrTotalCounterEnergy_Consumption;
END_IF

//EM8 (CEE32 3phase Measurement)
fbEM8(
	bEnable:= TRUE, 
	bChannel1Invers:= FALSE,
	bChannel2Invers:= FALSE,
	bChannel3Invers:= FALSE,
	uiCurrentTransformerRatioL1:= 35, 
	uiCurrentTransformerRatioL2:= 35, 
	uiCurrentTransformerRatioL3:= 35, 
	uiKBusState_IN:= fbKBusState.uiKBusState_OUT, 
	stDataEMPower=> , 
	stDataEMCounter=> , 
	stDataEMPowerRealTime=> , 
	stDataEMCounterRealTime=> , 
	diNrOfEM_OUT=> );

lr_RealPower_EM8 := fbEM8.stDataEMPower.lrPowerTotal;
lr_ApparentPower_EM8 := fbEM8.stDataEMPower.lrApparentPowerTotal;
lr_ReactivePower_EM8 := fbEM8.stDataEMPower.lrReactivePowerTotal;
lr_Frequency_EM8 := fbEM8.stDataEMPower.lrFrequency;
lr_RealPower_EM8_L1 := fbEM8.stDataEMPower.lrPowerL1;
lr_RealPower_EM8_L2 := fbEM8.stDataEMPower.lrPowerL2;
lr_RealPower_EM8_L3 := fbEM8.stDataEMPower.lrPowerL3;
lr_Voltage_EM8_L1N := fbEM8.stDataEMPower.lrVoltageL1N;
lr_Voltage_EM8_L2N := fbEM8.stDataEMPower.lrVoltageL2N;
lr_Voltage_EM8_L3N := fbEM8.stDataEMPower.lrVoltageL3N;
lr_Voltage_EM8_L1L2 := fbEM8.stDataEMPower.lrVoltageL1L2;
lr_Voltage_EM8_L2L3 := fbEM8.stDataEMPower.lrVoltageL2L3;
lr_Voltage_EM8_L3L1 := fbEM8.stDataEMPower.lrVoltageL3L1;
lr_Current_EM8_L1 := fbEM8.stDataEMPower.lrCurrentL1;
lr_Current_EM8_L2 := fbEM8.stDataEMPower.lrCurrentL2;
lr_Current_EM8_L3 := fbEM8.stDataEMPower.lrCurrentL3;
lr_Powerfactor_EM8_L1 := fbEM8.lrPowerfactorL1;
lr_Powerfactor_EM8_L2 := fbEM8.lrPowerfactorL2;
lr_Powerfactor_EM8_L3 := fbEM8.lrPowerfactorL3;
(*
lr_ApparentPower_EM8_L1 := fbEM8.lrApparentPowerL1;
lr_ApparentPower_EM8_L2 := fbEM8.lrApparentPowerL2;
lr_ApparentPower_EM8_L3 := fbEM8.lrApparentPowerL3;
lr_ReactivePower_EM8_L1 := fbEM8.lrReactivePowerL1;
lr_ReactivePower_EM8_L2 := fbEM8.lrReactivePowerL2;
lr_ReactivePower_EM8_L3 := fbEM8.lrReactivePowerL3;
*)
fbEM8Counter(
	byActiveTariff:= 1, 
	lrPowerInput:= lr_RealPower_EM8, 
	lrTotalCounterEnergy_Consumption=> , 
	lrTotalCounterEnergy_Production=> , 
	lrCounterEnergyT1_Consumption=> , 
	lrCounterEnergyT2_Consumption=> , 
	lrCounterEnergyT1_Production=> , 
	lrCounterEnergyT2_Production=> );
	
IF fbEM8Counter.lrTotalCounterEnergy_Consumption > lr_EnergyCounter_EM8 THEN  	
	lr_EnergyCounter_EM8 := fbEM8Counter.lrTotalCounterEnergy_Consumption;
END_IF

//EM9 (CEE32 3phase Measurement)
fbEM9(
	bEnable:= TRUE, 
	bChannel1Invers:= FALSE,
	bChannel2Invers:= FALSE,
	bChannel3Invers:= FALSE,
	uiCurrentTransformerRatioL1:= 35, 
	uiCurrentTransformerRatioL2:= 35, 
	uiCurrentTransformerRatioL3:= 35, 
	uiKBusState_IN:= fbKBusState.uiKBusState_OUT, 
	stDataEMPower=> , 
	stDataEMCounter=> , 
	stDataEMPowerRealTime=> , 
	stDataEMCounterRealTime=> , 
	diNrOfEM_OUT=> );

lr_RealPower_EM9 := fbEM9.stDataEMPower.lrPowerTotal;
lr_ApparentPower_EM9 := fbEM9.stDataEMPower.lrApparentPowerTotal;
lr_ReactivePower_EM9 := fbEM9.stDataEMPower.lrReactivePowerTotal;
lr_Frequency_EM9 := fbEM9.stDataEMPower.lrFrequency;
lr_RealPower_EM9_L1 := fbEM9.stDataEMPower.lrPowerL1;
lr_RealPower_EM9_L2 := fbEM9.stDataEMPower.lrPowerL2;
lr_RealPower_EM9_L3 := fbEM9.stDataEMPower.lrPowerL3;
lr_Voltage_EM9_L1N := fbEM9.stDataEMPower.lrVoltageL1N;
lr_Voltage_EM9_L2N := fbEM9.stDataEMPower.lrVoltageL2N;
lr_Voltage_EM9_L3N := fbEM9.stDataEMPower.lrVoltageL3N;
lr_Voltage_EM9_L1L2 := fbEM9.stDataEMPower.lrVoltageL1L2;
lr_Voltage_EM9_L2L3 := fbEM9.stDataEMPower.lrVoltageL2L3;
lr_Voltage_EM9_L3L1 := fbEM9.stDataEMPower.lrVoltageL3L1;
lr_Current_EM9_L1 := fbEM9.stDataEMPower.lrCurrentL1;
lr_Current_EM9_L2 := fbEM9.stDataEMPower.lrCurrentL2;
lr_Current_EM9_L3 := fbEM9.stDataEMPower.lrCurrentL3;
lr_Powerfactor_EM9_L1 := fbEM9.lrPowerfactorL1;
lr_Powerfactor_EM9_L2 := fbEM9.lrPowerfactorL2;
lr_Powerfactor_EM9_L3 := fbEM9.lrPowerfactorL3;
(*
lr_ApparentPower_EM9_L1 := fbEM9.lrApparentPowerL1;
lr_ApparentPower_EM9_L2 := fbEM9.lrApparentPowerL2;
lr_ApparentPower_EM9_L3 := fbEM9.lrApparentPowerL3;
lr_ReactivePower_EM9_L1 := fbEM9.lrReactivePowerL1;
lr_ReactivePower_EM9_L2 := fbEM9.lrReactivePowerL2;
lr_ReactivePower_EM9_L3 := fbEM9.lrReactivePowerL3;
*)
fbEM9Counter(
	byActiveTariff:= 1, 
	lrPowerInput:= lr_RealPower_EM9, 
	lrTotalCounterEnergy_Consumption=> , 
	lrTotalCounterEnergy_Production=> , 
	lrCounterEnergyT1_Consumption=> , 
	lrCounterEnergyT2_Consumption=> , 
	lrCounterEnergyT1_Production=> , 
	lrCounterEnergyT2_Production=> );
	
IF fbEM9Counter.lrTotalCounterEnergy_Consumption > lr_EnergyCounter_EM9 THEN  	
	lr_EnergyCounter_EM9 := fbEM9Counter.lrTotalCounterEnergy_Consumption;
END_IF

END_PROGRAM

// ---- FBs/FB_EM_Beckhoff_KL3403_T.TcPOU
FUNCTION_BLOCK FB_EM_Beckhoff_KL3403_T
VAR_INPUT PERSISTENT
	bEnable							: BOOL;											//Enable the function
	bChannel1Invers					: BOOL;											//Invert the Output data from Channel 1. = L1
	bChannel2Invers					: BOOL;											//Invert the Output data from Channel 2. = L2
	bChannel3Invers					: BOOL;											//Invert the Output data from Channel 3. = L3
	uiCurrentTransformerRatioL1		: UINT;											//Current Transformer Ratio for Channel 1 (L1)
	uiCurrentTransformerRatioL2		: UINT;											//Current Transformer Ratio for Channel 2 (L2)
	uiCurrentTransformerRatioL3		: UINT;											//Current Transformer Ratio for Channel 3 (L3)
END_VAR
VAR_INPUT
	uiKBusState_IN					: UINT;											//K-Bus State from the K-Bus Box on wich the Terminal is connected. (Connect with FB_K_Bus_state)
END_VAR
VAR_OUTPUT
	stDataEMPower					: ST_ElectricMeter_Output_Power;				//Output structure with Data from Electric Meter (Power Data)
	stDataEMCounter					: ST_ElectricMeter_Output_Counter;				//Output structure with Data from Electric Meter (Counter Data)
	stDataEMPowerRealTime			: ST_ElectricMeter_Output_Power;				//Output structure with Data from Electric Meter (Power Data RealTime)
	stDataEMCounterRealTime			: ST_ElectricMeter_Output_Counter;				//Output structure with Data from Electric Meter (Counter Data RealTime)
	diNrOfEM_OUT					: DINT;											//Active Number from the Electric Meter for using on other functions
	lrPowerfactorL1					: LREAL;
	lrPowerfactorL2					: LREAL;
	lrPowerfactorL3					: LREAL;
	lrApparentPowerL1				: LREAL;
	lrApparentPowerL2				: LREAL;
	lrApparentPowerL3				: LREAL;
	lrReactivePowerL1				: LREAL;
	lrReactivePowerL2				: LREAL;
	lrReactivePowerL3				: LREAL;
END_VAR
VAR
	{attribute 'conditionalshow'}
	fbEM							: FB_ElectricMeter;								//Electric Meter Function
	{attribute 'conditionalshow'}
	fbEnergyCounter					: FB_EnergyCounter;								//FB energy Counter, because the KL3403 has no nice logic for the Energy value
	{attribute 'hide'}
	fbNumberDevice					: FB_NumberOfDevice;							//Function block to calcualte the number of the Device
	fbKL3403						: FB_KL3403_SimpleProcessImage;					//Function KL3403
	{attribute 'hide'}
	stDataL1						: ST_KL3403;									//Data from Channel 1 (L1)
	{attribute 'hide'}
	stDataL2						: ST_KL3403;									//Data from Channel 2 (L2)
	{attribute 'hide'}
	stDataL3						: ST_KL3403;									//Data from Channel 3 (L3)
	{attribute 'hide'}
	timDissableFunctions			: TON;											//Timer to dissable the Function after Lynus_Standards.Constants_General.tTimeDissableLynusFunctions Days without connection to the Lynus Cloud
	{attribute 'hide'}
	timResetConnectionOnGVL			: TON;											//Timer to try reset the connection Flag on the GVL. (When somebody delete the Connection Function and make only a onlinechange)
	{attribute 'hide'}
	timSetCounterValues				: TON;											//Timer to set the counter values from the KL3403 Function to the EM Function
	{attribute 'hide'}
	arrPD							: ARRAY[1..7] OF FB_PersistentData_Number;		//Function to save persistent data
	{attribute 'hide'}
	byWaitInStep					: BYTE;											//Wait in Step before start to clean data on PLC
	{attribute 'hide'}
	iStateGVLData					: INT;											//State machine to handle the data on the GVL
	{attribute 'hide'}
	diCounterForGVL					: DINT;											//Counter to clean old data on GVL
END_VAR

//Creator : Kai Ebensperger
//Company : Lynus AG
//Date : 04.10.2021
//Version : 1.0.0.0

//Stefan: Addes S and Q calculation

//With this function is possible to read out all Information from a KL3403
//This Function support only the Simple Process Image and the Ratio in the Terminal register must be Set allways to 1.

//NOTE for diNr.....Designation => 
//_IN = Here Data come in from other Functions or go out to other functions about the GVL
//_OUT = Here Data go out to other functions about the GVL

(*-------------------------------------------------------------Calcualte the number of EM---------------------------------------------------------------*)

fbNumberDevice(
	diActualNumberOfDevices:= Lynus_Standards.GVL_Energy.stNumberOfDevices.diNumberOfElectricMeters, 
	diMaxNumberOfDevices:= Constants_Energy.diMaxNumberOfElectricMeters, 
	udiCounterOnlineChange:= TwinCAT_SystemInfoVarList._AppInfo.OnlineChangeCnt, 
	bNumberIsCalculatet=> , 
	bFPNumberIsCalculatet=> , 
	bOnlineChange=> , 
	diNumberForThisDevice=> diNrOfEM_OUT, 
	diNumberOfTotalDevices=> );

//Write new Numer on GVL
IF fbNumberDevice.bFPNumberIsCalculatet THEN
	Lynus_Standards.GVL_Energy.stNumberOfDevices.diNumberOfElectricMeters := fbNumberDevice.diNumberOfTotalDevices;	
END_IF

//Delete old Number on GVL
IF fbNumberDevice.bOnlineChange THEN 
	Lynus_Standards.GVL_Energy.stNumberOfDevices.diNumberOfElectricMeters := diNrOfEM_OUT;	
		iStateGVLData := 1; 
END_IF

(*-------------------------------------------------------------Service from Backend is ready and check the connection to backen for dissabel/enable Function---------------------------------------------------------------*)

//Try to reset the variable for connection on the GVL. When all is normal then the Lynus Mqtt connection function set this variable to true in the next cycle
//When we have no connection to the backend then after Lynus_Standards.Constants_General.tTimeDissableLynusFunctions days the Function is dissabled with all of his functionalities
timResetConnectionOnGVL(IN:= NOT timResetConnectionOnGVL.Q, PT:= T#1H, Q=> , ET=> );
	IF timResetConnectionOnGVL.Q THEN Lynus_Standards.GVL_Communicator.bStateConnectionToEnableFunctions := FALSE; END_IF
		IF NOT Lynus_Standards.GVL_Communicator.bStateConnectionToEnableFunctions THEN timDissableFunctions.IN := TRUE; ELSE timDissableFunctions.IN := FALSE; END_IF  
			timDissableFunctions(IN:= , PT:= Lynus_Standards.Constants_General.tTimeDissableLynusFunctions, Q=> , ET=> );

(*----------------------------------------------------------------------------------------KL3403 Communication----------------------------------------------------------------------------------------------*)

fbKL3403(
	uiKBusState_IN:= uiKBusState_IN, 
	uiCurrentTransformerRatioL1:= uiCurrentTransformerRatioL1,
	uiCurrentTransformerRatioL2:= uiCurrentTransformerRatioL2,
	uiCurrentTransformerRatioL3:= uiCurrentTransformerRatioL3,
	rResolutionCurrent:= 0.001,
	rResolutionPower:= 0.1,
	rResolutionEnergy:= 0.01,
	stDataL1=> , 
	stDataL2=> ,
	stDataL3=> );

//Invert the Output data, because it is possible that the current transformers have been mounted in different mounting positions.
IF NOT bChannel1Invers THEN
	stDataL1 := fbKL3403.stDataL1;
ELSE
	stDataL1.byErrorWarning := fbKL3403.stDataL1.byErrorWarning;
	stDataL1.rCurrent := fbKL3403.stDataL1.rCurrent;
	stDataL1.rVoltage := fbKL3403.stDataL1.rVoltage;
	stDataL1.rPower := fbKL3403.stDataL1.rPower * - 1;
	stDataL1.rPowerfactor := fbKL3403.stDataL1.rPowerfactor;
	stDataL1.rEnergy := fbKL3403.stDataL1.rEnergy;
	stDataL1.rFrequency := fbKL3403.stDataL1.rFrequency;
	stDataL1.rPeakValueCurrent := fbKL3403.stDataL1.rPeakValueCurrent;
	stDataL1.rPeakValueVoltage := fbKL3403.stDataL1.rPeakValueVoltage;
	stDataL1.rPeakValuePower := fbKL3403.stDataL1.rPeakValuePower * - 1;
	stDataL1.rMinValueCurrent := fbKL3403.stDataL1.rMinValueCurrent;
	stDataL1.rMinValueVoltage := fbKL3403.stDataL1.rMinValueVoltage;
	stDataL1.rMinValuePower := fbKL3403.stDataL1.rMinValuePower * - 1;
END_IF

IF NOT bChannel2Invers THEN
	stDataL2 := fbKL3403.stDataL2;
ELSE
	stDataL2.byErrorWarning := fbKL3403.stDataL2.byErrorWarning;
	stDataL2.rCurrent := fbKL3403.stDataL2.rCurrent;
	stDataL2.rVoltage := fbKL3403.stDataL2.rVoltage;
	stDataL2.rPower := fbKL3403.stDataL2.rPower * - 1;
	stDataL2.rPowerfactor := fbKL3403.stDataL2.rPowerfactor;
	stDataL2.rEnergy := fbKL3403.stDataL2.rEnergy;
	stDataL2.rFrequency := fbKL3403.stDataL2.rFrequency;
	stDataL2.rPeakValueCurrent := fbKL3403.stDataL2.rPeakValueCurrent;
	stDataL2.rPeakValueVoltage := fbKL3403.stDataL2.rPeakValueVoltage;
	stDataL2.rPeakValuePower := fbKL3403.stDataL2.rPeakValuePower * - 1;
	stDataL2.rMinValueCurrent := fbKL3403.stDataL2.rMinValueCurrent;
	stDataL2.rMinValueVoltage := fbKL3403.stDataL2.rMinValueVoltage;
	stDataL2.rMinValuePower := fbKL3403.stDataL2.rMinValuePower * - 1;
END_IF

IF NOT bChannel3Invers THEN
	stDataL3 := fbKL3403.stDataL3;
ELSE
	stDataL3.byErrorWarning := fbKL3403.stDataL3.byErrorWarning;
	stDataL3.rCurrent := fbKL3403.stDataL3.rCurrent;
	stDataL3.rVoltage := fbKL3403.stDataL3.rVoltage;
	stDataL3.rPower := fbKL3403.stDataL3.rPower * - 1;
	stDataL3.rPowerfactor := fbKL3403.stDataL3.rPowerfactor;
	stDataL3.rEnergy := fbKL3403.stDataL3.rEnergy;
	stDataL3.rFrequency := fbKL3403.stDataL3.rFrequency;
	stDataL3.rPeakValueCurrent := fbKL3403.stDataL3.rPeakValueCurrent;
	stDataL3.rPeakValueVoltage := fbKL3403.stDataL3.rPeakValueVoltage;
	stDataL3.rPeakValuePower := fbKL3403.stDataL3.rPeakValuePower * - 1;
	stDataL3.rMinValueCurrent := fbKL3403.stDataL3.rMinValueCurrent;
	stDataL3.rMinValueVoltage := fbKL3403.stDataL3.rMinValueVoltage;
	stDataL3.rMinValuePower := fbKL3403.stDataL3.rMinValuePower * - 1;
END_IF
	
(*----------------------------------------------------------------------------------------Energy Counter Function----------------------------------------------------------------------------------------------*)

//For the KL3403 we use a external Energy Counter Function. So we can count Import and Export Energy with the KL3403.
//Attetntion, the KL3403 is not MID Conform. Thus, these values must not be used for billing.
fbEnergyCounter(
	byActiveTariff:= 1, 
	lrPowerInput:= (stDataL1.rPower + stDataL2.rPower + stDataL3.rPower) / 1000, 
	lrTotalCounterEnergy_Consumption=> , 
	lrTotalCounterEnergy_Production=> , 
	lrCounterEnergyT1_Consumption=> , 
	lrCounterEnergyT2_Consumption=> , 
	lrCounterEnergyT1_Production=> , 
	lrCounterEnergyT2_Production=> );

(*----------------------------------------------------------------------------------------Electric Meter Function----------------------------------------------------------------------------------------------*)

//Error
IF timDissableFunctions.Q THEN fbEM.bWarning := TRUE; fbEM.iWarningCode := 0; ELSE fbEM.bWarning := FALSE; END_IF 
	IF Lynus_Standards.GVL_Energy.stNumberOfDevices.diNumberOfElectricMeters > Constants_Energy.diMaxNumberOfElectricMeters OR 
		stDataL1.byErrorWarning = 2 OR stDataL2.byErrorWarning = 2 OR stDataL3.byErrorWarning = 2 THEN 
			fbEM.bError := TRUE; 
	ELSE 
			fbEM.bError := FALSE; 
	END_IF
		IF Lynus_Standards.GVL_Energy.stNumberOfDevices.diNumberOfElectricMeters > Constants_Energy.diMaxNumberOfElectricMeters THEN fbEM.iErrorCode := 1;
		ELSIF stDataL1.byErrorWarning = 2 OR stDataL2.byErrorWarning = 2 OR stDataL3.byErrorWarning = 2 THEN fbEM.iErrorCode := 0;
		END_IF

timSetCounterValues(IN:= bEnable AND NOT timSetCounterValues.Q, PT:= T#2S, Q=> , ET=> );		

//Function
fbEM(
	bEnable:= bEnable AND NOT timDissableFunctions.Q, 
	bError:= , 
	bEnableReadOutFunction:= FALSE, 
	bWriteWithDelay:= TRUE, 
	bPowerDataInvers:= FALSE,
	bReadOutDataDone:= timSetCounterValues.Q,
	iTimeReadOutInterval:= 0, 
	iErrorCode:= , 
	iWarningCode:= , 
	lrTotalCounterEnergy_Consumption:= fbEnergyCounter.lrTotalCounterEnergy_Consumption,
	lrTotalCounterEnergy_Production:= fbEnergyCounter.lrTotalCounterEnergy_Production, 
	lrCounterEnergyT1_Consumption:= fbEnergyCounter.lrCounterEnergyT1_Consumption,
	lrCounterEnergyT2_Consumption:= fbEnergyCounter.lrCounterEnergyT2_Consumption,
	lrCounterEnergyT1_Production:= fbEnergyCounter.lrCounterEnergyT1_Production, 
	lrCounterEnergyT2_Production:= fbEnergyCounter.lrCounterEnergyT2_Production, 
	lrCurrentL1:= stDataL1.rCurrent, 
	lrVoltageL1N:= stDataL1.rVoltage, 
	lrVoltageL1L2:= stDataL1.rVoltage*SQRT(3), 
	lrPowerL1:= stDataL1.rPower, 
	lrCurrentL2:= stDataL2.rCurrent, 
	lrVoltageL2N:= stDataL2.rVoltage, 
	lrVoltageL2L3:= stDataL2.rVoltage*SQRT(3), 
	lrPowerL2:= stDataL2.rPower, 
	lrCurrentL3:= stDataL3.rCurrent, 
	lrVoltageL3N:= stDataL3.rVoltage, 
	lrVoltageL3L1:= stDataL3.rVoltage*SQRT(3), 
	lrPowerL3:= stDataL3.rPower, 
	lrPowerTotal:= stDataL1.rPower + stDataL2.rPower + stDataL3.rPower, 
	lrFrequency:= (stDataL1.rFrequency + stDataL2.rFrequency + stDataL3.rFrequency) / 3, 
 	lrApparentPowerTotal:=,
	lrReactivePowerTotal:=, 
	tTimDelayOutput:= T#5S, 
	stDataEMOutPower=> stDataEMPowerRealTime, 
	stDataEMOutPowerDelay=> stDataEMPower, 
	stDataEMOutCounter=> stDataEMCounterRealTime,
	stDataEMOutCounterDelay=> stDataEMCounter,
	bReadOutMeter=> );


	//calculate total apparant power in VA
	fbEM.lrApparentPowerTotal := fbEM.lrVoltageL1N * fbEM.lrCurrentL1 + fbEM.lrVoltageL2N * fbEM.lrCurrentL2 +  fbEM.lrVoltageL3N * fbEM.lrCurrentL3;
	
	IF fbEM.lrApparentPowerTotal<>0 AND fbEM.lrPowerTotal<>0 AND fbEM.lrApparentPowerTotal> ABS(fbEM.lrPowerTotal) THEN
		fbEM.lrReactivePowerTotal:= SQRT(ABS(fbEM.lrApparentPowerTotal*fbEM.lrApparentPowerTotal - ABS(fbEM.lrPowerTotal*fbEM.lrPowerTotal)));	
	END_IF
	IF stDataL1.rPowerfactor<>0 AND stDataL2.rPowerfactor <>0 AND stDataL3.rPowerfactor<>0 THEN 	// check that not all cos phi are not 0
		IF (stDataL1.rPowerfactor+stDataL2.rPowerfactor+stDataL3.rPowerfactor)<>0 THEN				// check that the sum is not 0	
			IF 	(stDataL1.rPowerfactor+stDataL2.rPowerfactor+stDataL3.rPowerfactor)/3<0 THEN		// check is the average is below 0 / capacitive
				fbEM.lrReactivePowerTotal:=fbEM.lrReactivePowerTotal*(-1);
			END_IF
		END_IF	
	END_IF
	
	//added Powerfactor output
	lrPowerfactorL1 := stDataL1.rPowerfactor;
	lrPowerfactorL2 := stDataL2.rPowerfactor;
	lrPowerfactorL3 := stDataL3.rPowerfactor;
	
	//added Apparent Power per Phase output
	lrApparentPowerL1 := (fbEM.lrVoltageL1N * fbEM.lrCurrentL1) / 1000;
	lrApparentPowerL2 := (fbEM.lrVoltageL2N * fbEM.lrCurrentL2) / 1000;
	lrApparentPowerL3 := (fbEM.lrVoltageL3N * fbEM.lrCurrentL3) / 1000;
	
	//added Reactive Power per Phase output
	lrReactivePowerL1 := SQRT(ABS(lrApparentPowerL1*lrApparentPowerL1 - ABS(fbEM.lrPowerL1 *fbEM.lrPowerL1))) / 1000;
	lrReactivePowerL2 := SQRT(ABS(lrApparentPowerL2*lrApparentPowerL2 - ABS(fbEM.lrPowerL2 *fbEM.lrPowerL2))) / 1000;
	lrReactivePowerL3 := SQRT(ABS(lrApparentPowerL3*lrApparentPowerL3 - ABS(fbEM.lrPowerL3 *fbEM.lrPowerL3))) / 1000;
	
(*-----------------------------------------------------------Handle data to Global structure for Electric Meter-----------------------------------------------------------------*)

CASE iStateGVLData OF
	
	0://Init Step
		byWaitInStep := 0;
			diCounterForGVL := 1;
	
	1://Wait for 4 Steps before clean al Data on GVL
		byWaitInStep := byWaitInStep + 1;
			IF byWaitInStep >= 4 AND fbNumberDevice.bNumberIsCalculatet THEN iStateGVLData := 2; END_IF
				//To much Devices, back to the Init step
				IF byWaitInStep >= 4 AND NOT fbNumberDevice.bNumberIsCalculatet THEN iStateGVLData := 0; END_IF	
			
	2://Clear all Data in GVL
		Lynus_Standards.GVL_Energy.stDataElectricMeters[diCounterForGVL].bEnabled := FALSE;	
			Lynus_Standards.GVL_Energy.stDataElectricMeters[diCounterForGVL].byErrorWarning := 0;
				Lynus_Standards.GVL_Energy.stDataElectricMeters[diCounterForGVL].lrCounterEnergyT1_Consumption := 0;
					Lynus_Standards.GVL_Energy.stDataElectricMeters[diCounterForGVL].lrCounterEnergyT1_Production := 0;
						Lynus_Standards.GVL_Energy.stDataElectricMeters[diCounterForGVL].lrCounterEnergyT2_Consumption := 0;
							Lynus_Standards.GVL_Energy.stDataElectricMeters[diCounterForGVL].lrCounterEnergyT2_Production := 0;
								Lynus_Standards.GVL_Energy.stDataElectricMeters[diCounterForGVL].lrPower := 0;
									Lynus_Standards.GVL_Energy.stDataElectricMeters[diCounterForGVL].lrPowerConsumption := 0;
										Lynus_Standards.GVL_Energy.stDataElectricMeters[diCounterForGVL].lrPowerProduction := 0;
											Lynus_Standards.GVL_Energy.stDataElectricMeters[diCounterForGVL].lrTotalCounterEnergy_Consumption := 0;
												Lynus_Standards.GVL_Energy.stDataElectricMeters[diCounterForGVL].lrTotalCounterEnergy_Production := 0;
		
		//Electric Meters
		diCounterForGVL := diCounterForGVL + 1;
			diCounterForGVL := LIMIT(0,diCounterForGVL,Constants_Energy.diMaxNumberOfElectricMeters);
				//Back to the init step
				IF diCounterForGVL >= Constants_Energy.diMaxNumberOfElectricMeters THEN iStateGVLData := 0; END_IF

END_CASE 	 

//Write Data on GVL for Electric Meter
IF diNrOfEM_OUT > 0 AND fbNumberDevice.bNumberIsCalculatet THEN
	Lynus_Standards.GVL_Energy.stDataElectricMeters[diNrOfEM_OUT].bEnabled := fbEM.stDataEMOutPower.bEnabled;
		Lynus_Standards.GVL_Energy.stDataElectricMeters[diNrOfEM_OUT].byErrorWarning := fbEM.stDataEMOutPower.byErrorWarning;
			Lynus_Standards.GVL_Energy.stDataElectricMeters[diNrOfEM_OUT].lrCounterEnergyT1_Consumption := fbEM.stDataEMOutCounter.lrCounterEnergyT1_Consumption;
				Lynus_Standards.GVL_Energy.stDataElectricMeters[diNrOfEM_OUT].lrCounterEnergyT1_Production := fbEM.stDataEMOutCounter.lrCounterEnergyT1_Production;
					Lynus_Standards.GVL_Energy.stDataElectricMeters[diNrOfEM_OUT].lrCounterEnergyT2_Consumption := fbEM.stDataEMOutCounter.lrCounterEnergyT2_Consumption;
						Lynus_Standards.GVL_Energy.stDataElectricMeters[diNrOfEM_OUT].lrCounterEnergyT2_Production := fbEM.stDataEMOutCounter.lrCounterEnergyT2_Production;		
							Lynus_Standards.GVL_Energy.stDataElectricMeters[diNrOfEM_OUT].lrPower := fbEM.stDataEMOutPower.lrPowerTotal;
								Lynus_Standards.GVL_Energy.stDataElectricMeters[diNrOfEM_OUT].lrPowerConsumption := fbEM.stDataEMOutPower.lrPowerConsumption;
									Lynus_Standards.GVL_Energy.stDataElectricMeters[diNrOfEM_OUT].lrPowerProduction := fbEM.stDataEMOutPower.lrPowerProduction;
										Lynus_Standards.GVL_Energy.stDataElectricMeters[diNrOfEM_OUT].lrTotalCounterEnergy_Consumption := fbEM.stDataEMOutCounter.lrTotalCounterEnergy_Consumption;
											Lynus_Standards.GVL_Energy.stDataElectricMeters[diNrOfEM_OUT].lrTotalCounterEnergy_Production := fbEM.stDataEMOutCounter.lrTotalCounterEnergy_Production;
END_IF

(*----------------------------------------------------------Save persistent data----------------------------------------------------------------*)

arrPD[1](lrValue:= BOOL_TO_LREAL(bEnable), bEventBasedActive=> );
arrPD[2](lrValue:= UINT_TO_LREAL(uiCurrentTransformerRatioL1), bEventBasedActive=> );
arrPD[3](lrValue:= UINT_TO_LREAL(uiCurrentTransformerRatioL2), bEventBasedActive=> );
arrPD[4](lrValue:= UINT_TO_LREAL(uiCurrentTransformerRatioL3), bEventBasedActive=> );
arrPD[5](lrValue:= BOOL_TO_LREAL(bChannel1Invers), bEventBasedActive=> );
arrPD[6](lrValue:= BOOL_TO_LREAL(bChannel2Invers), bEventBasedActive=> );
arrPD[7](lrValue:= BOOL_TO_LREAL(bChannel3Invers), bEventBasedActive=> );

END_FUNCTION_BLOCK

// ---- POUs/prgCalc.TcPOU
PROGRAM prgCalc
VAR
	//Sum of all CEE32 Measurements
	fbEMTotalCounter		: FB_EnergyCounter;
	lr_RealPower_Total		: LREAL;					//{#lynus.ag#()}
END_VAR

VAR PERSISTENT
	lr_EnergyCounter_Total	: LREAL;					//{#lynus.ag#()}
END_VAR


lr_RealPower_Total := 	prgEM.lr_RealPower_EM1 + 
						prgEM.lr_RealPower_EM2 + 
						prgEM.lr_RealPower_EM3 + 
						prgEM.lr_RealPower_EM4 + 
						prgEM.lr_RealPower_EM5 + 
						prgEM.lr_RealPower_EM6 + 
						prgEM.lr_RealPower_EM7 + 
						prgEM.lr_RealPower_EM8 + 
						prgEM.lr_RealPower_EM9;

fbEMTotalCounter(
	byActiveTariff:= 1, 
	lrPowerInput:= lr_RealPower_Total, 
	lrTotalCounterEnergy_Consumption=> , 
	lrTotalCounterEnergy_Production=> , 
	lrCounterEnergyT1_Consumption=> , 
	lrCounterEnergyT2_Consumption=> , 
	lrCounterEnergyT1_Production=> , 
	lrCounterEnergyT2_Production=> );
	
IF fbEMTotalCounter.lrTotalCounterEnergy_Consumption > lr_EnergyCounter_Total THEN  	
	lr_EnergyCounter_Total := fbEMTotalCounter.lrTotalCounterEnergy_Consumption;
END_IF

END_PROGRAM

// ---- POUs/prgComEffIO.TcPOU
PROGRAM prgComEffIO
VAR
	fbCom		: FB_MqttCommunicator_V2;
	int_SSPNumber: INT;
END_VAR

fbCom(
	bConnect:= TRUE, 
	strAuthKey:= 'EIO08031879806', 
	sUserName:= , 
	sUserPassword:= , 
	eSavePositionCertificate:= eSavePositionOnPLC.ePostionHardDisk,  
	bConnected=> , 
	bError=> , 
	hrErrorCode=> , 
	eConnectionState=> , 
	eErrorMessage_Out=> );


prg_ReadDeviceName();
IF prg_ReadDeviceName.sDeviceName = '' THEN
	prg_ReadDeviceName.bStart := TRUE;
END_IF


// select user / pass according device name:

IF prg_ReadDeviceName.sDeviceName = 'EIOSV010001' THEN
	fbCom.sUserName:= 'e9f67ebc-f8a4-4bb2-949c-26b68dda2543'; 
    fbCom.sUserPassword:= '0685927c-b6f6-4802-a1d9-1256766da196';
	int_SSPNumber :=1;
ELSIF prg_ReadDeviceName.sDeviceName = 'EIOSV010002' THEN
	fbCom.sUserName:= '88eb7225-2446-4047-be39-c50e45046d19'; 
    fbCom.sUserPassword:= '92f99f89-c875-4be9-825b-3430c234338c';
	int_SSPNumber :=2;
END_IF

END_PROGRAM
